FUNCTION_BLOCK PrintString
  (* Standard: 61499-2 *)
  (* Version 0.1, 2017-00-09, hpea485, UOA *)
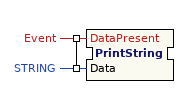
  EVENT_INPUT
    DataPresent WITH Data;
  END_EVENT
  VAR_INPUT
    Data : STRING;
  END_VAR
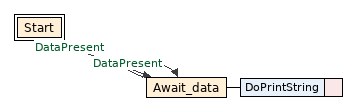
  EC_STATES
    Start;
    Await_data : DoPrintString;
  END_STATES
  EC_TRANSITIONS
    Start TO Await_data := DataPresent;
    Await_data TO Await_data := DataPresent;
  END_TRANSITIONS
  ALGORITHM DoPrintString IN C:
printf("PrintString: %s\n", me->Data);
  END_ALGORITHM
END_FUNCTION_BLOCK
